// TIA Portal V16 export
// export: Created 2021-11-12T13:32:33.9324246Z, ExportSetting WithDefaults, DisplayName Totally Integrated Automation Portal, DisplayVersion V16 Update 3, DisplayName TIA Portal Version Control Interface, DisplayVersion V16 Update 2, DisplayName TIA Portal Openness, DisplayVersion V16 Update 3, DisplayName SINAMICS Startdrive Advanced, DisplayVersion V16 Update 5, DisplayName SINAMICS Startdrive G130, G150, S120, S150, SINAMICS MV, S210, DisplayVersion V16 Update 5, DisplayName SINAMICS Startdrive G110M, G120, G120C, G120D, G120P, G115D, DisplayVersion V16 Update 5, DisplayName STEP 7 Professional, DisplayVersion V16 Update 3, DisplayName STEP 7 Safety, DisplayVersion V16, DisplayName WinCC UA Professional, DisplayVersion V16 Update 3
FUNCTION_BLOCK "Station220"   // FB16, LAD
{ S7_Optimized_Access := 'TRUE' }
VERSION : 0.1
// Dopravník na ostřižky
// stored: AutoNumber true, IsIECCheckEnabled false, IsRetainMemResEnabled false, MemoryReserve 100, SetENOAutomatically false, UDAEnableTagReadback false
   VAR
      SF_CL01_Alarm { S7_SetPoint := 'True'} : "STD_DI_Mon";
      SF_CL01_Warning { S7_SetPoint := 'True'} : "STD_DI_Mon";
      SF_GL01MA01 { S7_SetPoint := 'True'} : "STD_Drive1";
      SF_UC12TA01 { S7_SetPoint := 'True'} : "STD_Siemens_G120_CU240E_2_PN";
      SF_TON_1 { S7_SetPoint := 'True'} : TON_TIME;
      SF_TOF_1 { S7_SetPoint := 'True'} : TOF_TIME;
      SF_CL01 { S7_SetPoint := 'True'} : "STD_PartCounter";
      SS_Edge { S7_SetPoint := 'True'} : Array[0..15] of Bool;
      SB1BoxExchangeReq { S7_SetPoint := 'True'} : Bool;
   END_VAR
   VAR_TEMP
      TS_GL01MA01 : "UDT_DriveControl";
      TS_UC12TA01 : Struct
         ReqDir1 : Bool;   // Move in direction 1
         ReqDir2 : Bool;   // Move in direction 2
         AckErr : Bool;   // Acknowledge error
         SpeedSP : Real;   // Speed setpoint
      END_STRUCT;
      TB1PwrOK : Bool;
      TDINoOfParts : DInt;   // Number of parts to count
      TB1BoxFull : Bool;   // Box is full
      TB1CountPulse : Bool;
   END_VAR
   VAR_TEMP   // added for the SCL form of the ladder/FBD networks
      _w1 : Bool;
      _w2 : Bool;
      _w3 : Bool;
      _w4 : Bool;
   END_VAR
BEGIN

REGION Network 1: Clear temporary variables
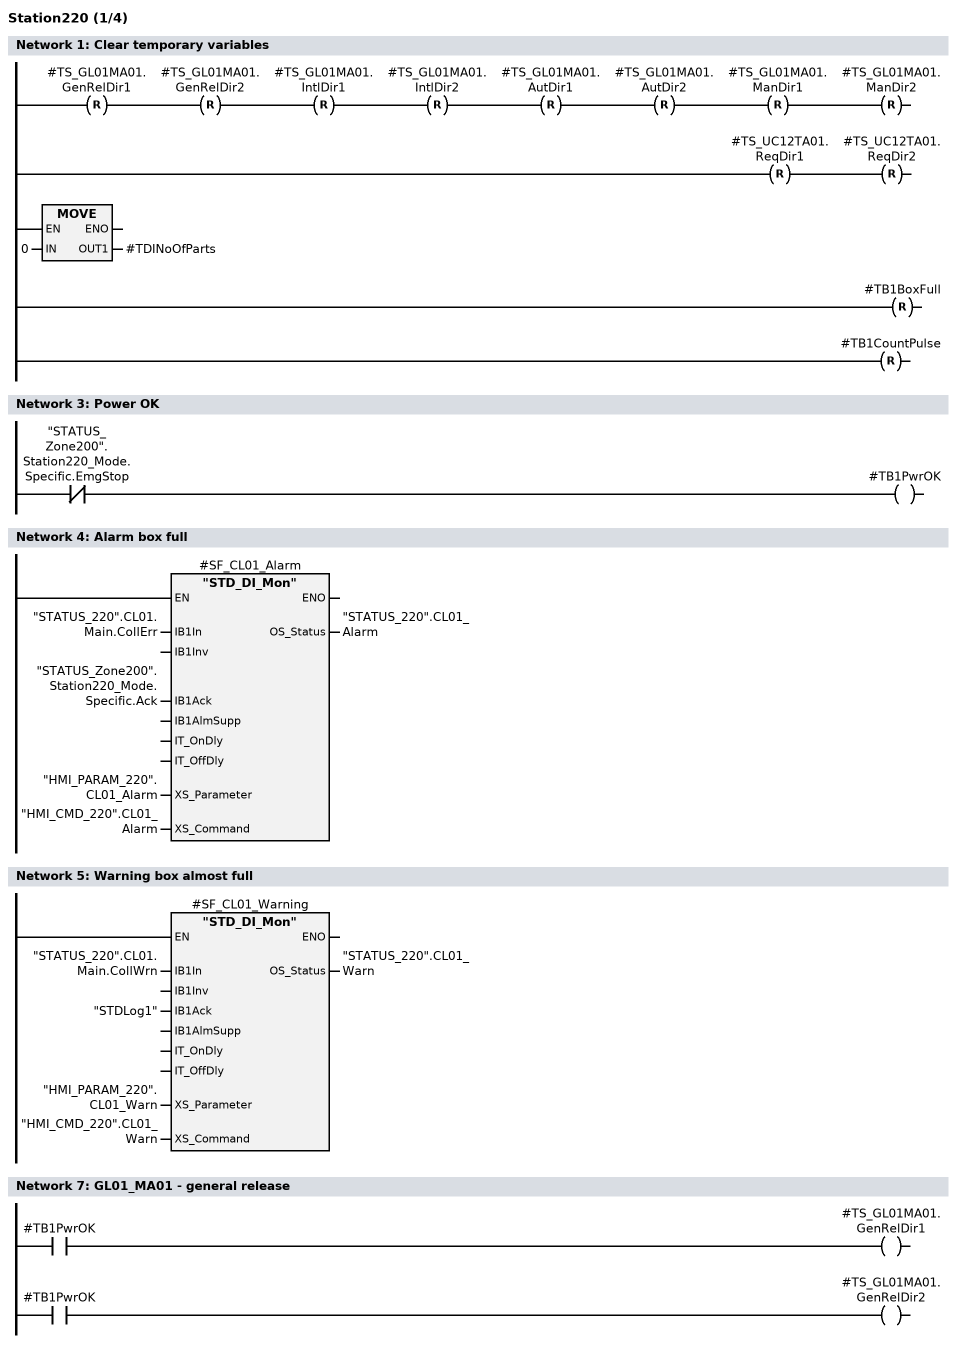
   RUNG wire#powerrail
      R_Coil( #TS_GL01MA01.GenRelDir1 )
      R_Coil( #TS_GL01MA01.GenRelDir2 )
      R_Coil( #TS_GL01MA01.IntlDir1 )
      R_Coil( #TS_GL01MA01.IntlDir2 )
      R_Coil( #TS_GL01MA01.AutDir1 )
      R_Coil( #TS_GL01MA01.AutDir2 )
      R_Coil( #TS_GL01MA01.ManDir1 )
      R_Coil( #TS_GL01MA01.ManDir2 )
   END_RUNG
   RUNG wire#powerrail
      R_Coil( #TS_UC12TA01.ReqDir1 )
      R_Coil( #TS_UC12TA01.ReqDir2 )
   END_RUNG
   RUNG wire#powerrail
      Move(in := 0, out1 => #TDINoOfParts)
   END_RUNG
   RUNG wire#powerrail
      R_Coil( #TB1BoxFull )
   END_RUNG
   RUNG wire#powerrail
      R_Coil( #TB1CountPulse )
   END_RUNG
   // the same network as SCL:
   #TS_GL01MA01.GenRelDir1 := FALSE;
   #TS_GL01MA01.GenRelDir2 := FALSE;
   #TS_GL01MA01.IntlDir1 := FALSE;
   #TS_GL01MA01.IntlDir2 := FALSE;
   #TS_GL01MA01.AutDir1 := FALSE;
   #TS_GL01MA01.AutDir2 := FALSE;
   #TS_GL01MA01.ManDir1 := FALSE;
   #TS_GL01MA01.ManDir2 := FALSE;
   #TS_UC12TA01.ReqDir1 := FALSE;
   #TS_UC12TA01.ReqDir2 := FALSE;
   #TDINoOfParts := 0;
   #TB1BoxFull := FALSE;
   #TB1CountPulse := FALSE;
END_REGION

REGION Network 2: *************** Alarms ***************
END_REGION

REGION Network 3: Power OK
   RUNG wire#powerrail
      I_Contact( "STATUS_Zone200".Station220_Mode.Specific.EmgStop )
      Coil( #TB1PwrOK )
   END_RUNG
   // the same network as SCL:
   #TB1PwrOK := NOT "STATUS_Zone200".Station220_Mode.Specific.EmgStop;
END_REGION

REGION Network 4: Alarm box full
   RUNG wire#powerrail
      #SF_CL01_Alarm(IB1In := "STATUS_220".CL01.Main.CollErr, IB1Inv :=, IB1Ack := "STATUS_Zone200".Station220_Mode.Specific.Ack, IB1AlmSupp :=, IT_OnDly :=, IT_OffDly :=, XS_Parameter := "HMI_PARAM_220".CL01_Alarm, XS_Command := "HMI_CMD_220".CL01_Alarm, OS_Status => "STATUS_220".CL01_Alarm)
   END_RUNG
   // the same network as SCL:
   #SF_CL01_Alarm(IB1In := "STATUS_220".CL01.Main.CollErr,   // "STD_DI_Mon"
                  IB1Ack := "STATUS_Zone200".Station220_Mode.Specific.Ack,
                  XS_Parameter := "HMI_PARAM_220".CL01_Alarm,
                  XS_Command := "HMI_CMD_220".CL01_Alarm,
                  OS_Status => "STATUS_220".CL01_Alarm);
END_REGION

REGION Network 5: Warning box almost full
   RUNG wire#powerrail
      #SF_CL01_Warning(IB1In := "STATUS_220".CL01.Main.CollWrn, IB1Inv :=, IB1Ack := "STDLog1", IB1AlmSupp :=, IT_OnDly :=, IT_OffDly :=, XS_Parameter := "HMI_PARAM_220".CL01_Warn, XS_Command := "HMI_CMD_220".CL01_Warn, OS_Status => "STATUS_220".CL01_Warn)
   END_RUNG
   // the same network as SCL:
   #SF_CL01_Warning(IB1In := "STATUS_220".CL01.Main.CollWrn,   // "STD_DI_Mon"
                    IB1Ack := "STDLog1",
                    XS_Parameter := "HMI_PARAM_220".CL01_Warn,
                    XS_Command := "HMI_CMD_220".CL01_Warn,
                    OS_Status => "STATUS_220".CL01_Warn);
END_REGION

REGION Network 6: *************** GL01_MA01 Conveyor drive ***************
END_REGION

REGION Network 7: GL01_MA01 - general release
   RUNG wire#powerrail
      Contact( #TB1PwrOK )
      Coil( #TS_GL01MA01.GenRelDir1 )
   END_RUNG
   RUNG wire#powerrail
      Contact( #TB1PwrOK )
      Coil( #TS_GL01MA01.GenRelDir2 )
   END_RUNG
   // the same network as SCL:
   #TS_GL01MA01.GenRelDir1 := #TB1PwrOK;
   #TS_GL01MA01.GenRelDir2 := #TB1PwrOK;
END_REGION

REGION Network 8: GL01_MA01 - interlocks
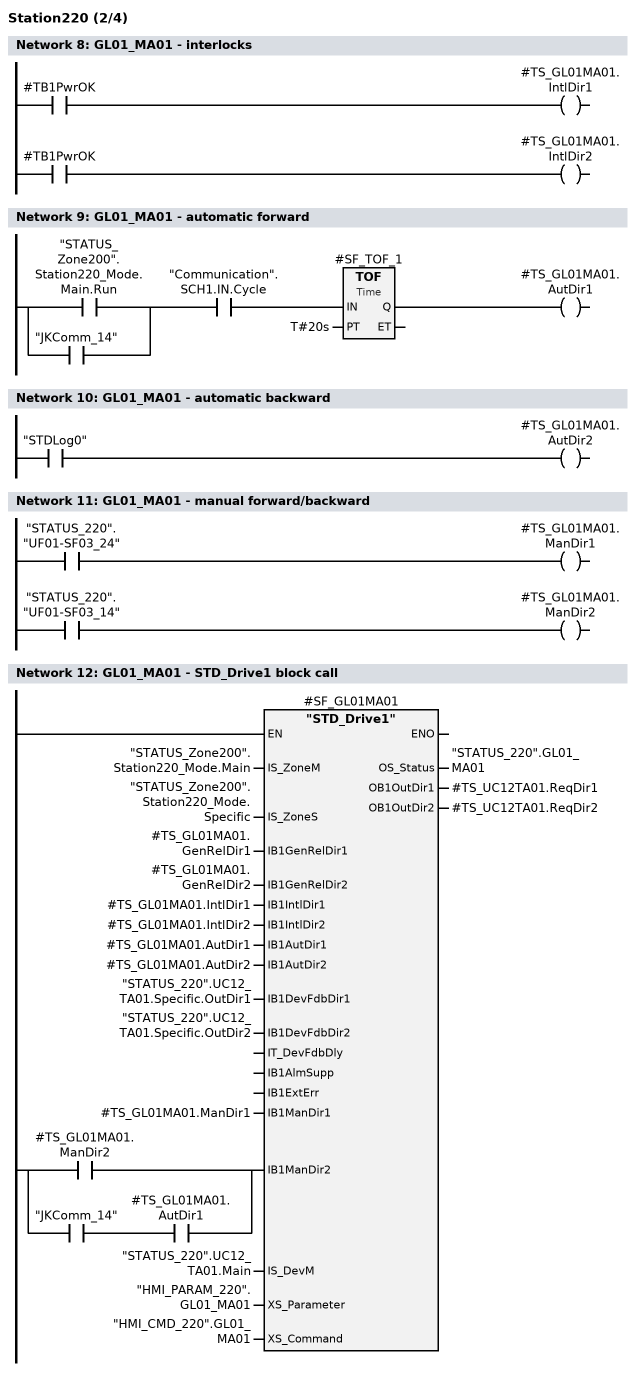
   RUNG wire#powerrail
      Contact( #TB1PwrOK )
      Coil( #TS_GL01MA01.IntlDir1 )
   END_RUNG
   RUNG wire#powerrail
      Contact( #TB1PwrOK )
      Coil( #TS_GL01MA01.IntlDir2 )
   END_RUNG
   // the same network as SCL:
   #TS_GL01MA01.IntlDir1 := #TB1PwrOK;
   #TS_GL01MA01.IntlDir2 := #TB1PwrOK;
END_REGION

REGION Network 9: GL01_MA01 - automatic forward
   RUNG wire#powerrail
      Contact( "STATUS_Zone200".Station220_Mode.Main.Run )
      wire#w1
      Contact( "Communication".SCH1.IN.Cycle )
      { S7_Templates := "time_type := Time" } #SF_TOF_1.TOF(pt := T#20s, et =>)
      Coil( #TS_GL01MA01.AutDir1 )
   END_RUNG
   RUNG wire#powerrail
      Contact( "JKComm_14" )
   END_RUNG wire#w1
   // the same network as SCL:
   #SF_TOF_1(IN := ("STATUS_Zone200".Station220_Mode.Main.Run OR "JKComm_14") AND "Communication".SCH1.IN.Cycle,   // TOF
             PT := T#20s);
   #TS_GL01MA01.AutDir1 := #SF_TOF_1.Q;
END_REGION

REGION Network 10: GL01_MA01 - automatic backward
   RUNG wire#powerrail
      Contact( "STDLog0" )
      Coil( #TS_GL01MA01.AutDir2 )
   END_RUNG
   // the same network as SCL:
   #TS_GL01MA01.AutDir2 := "STDLog0";
END_REGION

REGION Network 11: GL01_MA01 - manual forward/backward
   RUNG wire#powerrail
      Contact( "STATUS_220"."UF01-SF03_24" )
      Coil( #TS_GL01MA01.ManDir1 )
   END_RUNG
   RUNG wire#powerrail
      Contact( "STATUS_220"."UF01-SF03_14" )
      Coil( #TS_GL01MA01.ManDir2 )
   END_RUNG
   // the same network as SCL:
   #TS_GL01MA01.ManDir1 := "STATUS_220"."UF01-SF03_24";
   #TS_GL01MA01.ManDir2 := "STATUS_220"."UF01-SF03_14";
END_REGION

REGION Network 12: GL01_MA01 - STD_Drive1 block call
   RUNG wire#powerrail
      #SF_GL01MA01(IB1ManDir2 := wire#w1, IS_ZoneM := "STATUS_Zone200".Station220_Mode.Main, IS_ZoneS := "STATUS_Zone200".Station220_Mode.Specific, IB1GenRelDir1 := #TS_GL01MA01.GenRelDir1, IB1GenRelDir2 := #TS_GL01MA01.GenRelDir2, IB1IntlDir1 := #TS_GL01MA01.IntlDir1, IB1IntlDir2 := #TS_GL01MA01.IntlDir2, IB1AutDir1 := #TS_GL01MA01.AutDir1, IB1AutDir2 := #TS_GL01MA01.AutDir2, IB1DevFdbDir1 := "STATUS_220".UC12_TA01.Specific.OutDir1, IB1DevFdbDir2 := "STATUS_220".UC12_TA01.Specific.OutDir2, IT_DevFdbDly :=, IB1AlmSupp :=, IB1ExtErr :=, IB1ManDir1 := #TS_GL01MA01.ManDir1, IS_DevM := "STATUS_220".UC12_TA01.Main, XS_Parameter := "HMI_PARAM_220".GL01_MA01, XS_Command := "HMI_CMD_220".GL01_MA01, OS_Status => "STATUS_220".GL01_MA01, OB1OutDir1 => #TS_UC12TA01.ReqDir1, OB1OutDir2 => #TS_UC12TA01.ReqDir2)
   END_RUNG
   RUNG wire#powerrail
      Contact( #TS_GL01MA01.ManDir2 )
   END_RUNG wire#w1
   RUNG wire#powerrail
      Contact( "JKComm_14" )
      Contact( #TS_GL01MA01.AutDir1 )
   END_RUNG wire#w1
   // the same network as SCL:
   #SF_GL01MA01(IS_ZoneM := "STATUS_Zone200".Station220_Mode.Main,   // "STD_Drive1"
                IS_ZoneS := "STATUS_Zone200".Station220_Mode.Specific,
                IB1GenRelDir1 := #TS_GL01MA01.GenRelDir1,
                IB1GenRelDir2 := #TS_GL01MA01.GenRelDir2,
                IB1IntlDir1 := #TS_GL01MA01.IntlDir1,
                IB1IntlDir2 := #TS_GL01MA01.IntlDir2,
                IB1AutDir1 := #TS_GL01MA01.AutDir1,
                IB1AutDir2 := #TS_GL01MA01.AutDir2,
                IB1DevFdbDir1 := "STATUS_220".UC12_TA01.Specific.OutDir1,
                IB1DevFdbDir2 := "STATUS_220".UC12_TA01.Specific.OutDir2,
                IB1ManDir1 := #TS_GL01MA01.ManDir1,
                IB1ManDir2 := #TS_GL01MA01.ManDir2 OR ("JKComm_14" AND #TS_GL01MA01.AutDir1),
                IS_DevM := "STATUS_220".UC12_TA01.Main,
                XS_Parameter := "HMI_PARAM_220".GL01_MA01,
                XS_Command := "HMI_CMD_220".GL01_MA01,
                OS_Status => "STATUS_220".GL01_MA01,
                OB1OutDir1 => #TS_UC12TA01.ReqDir1,
                OB1OutDir2 => #TS_UC12TA01.ReqDir2);
END_REGION

REGION Network 13: UC12_TA01 - Acknowledge error
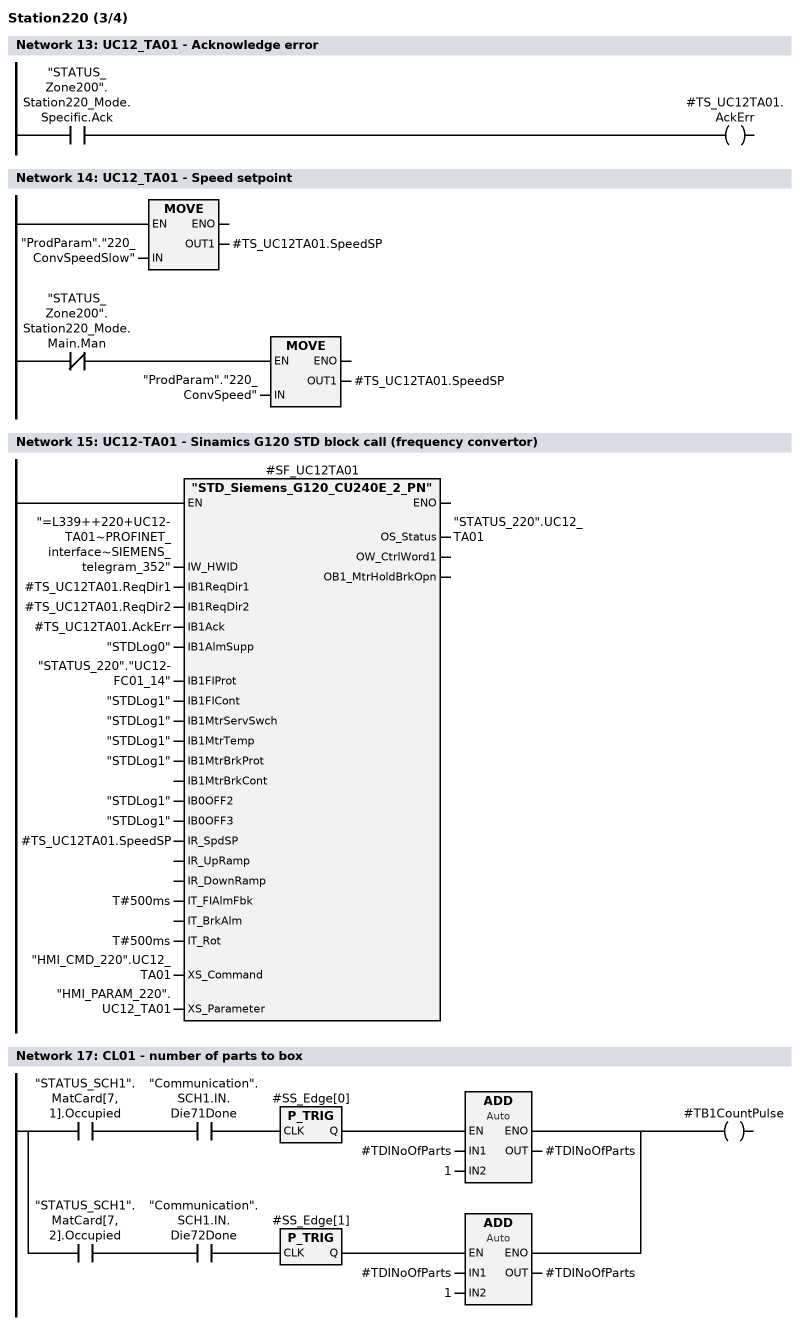
   RUNG wire#powerrail
      Contact( "STATUS_Zone200".Station220_Mode.Specific.Ack )
      Coil( #TS_UC12TA01.AckErr )
   END_RUNG
   // the same network as SCL:
   #TS_UC12TA01.AckErr := "STATUS_Zone200".Station220_Mode.Specific.Ack;
END_REGION

REGION Network 14: UC12_TA01 - Speed setpoint
   RUNG wire#powerrail
      Move(in := "ProdParam"."220_ConvSpeedSlow", out1 => #TS_UC12TA01.SpeedSP)
   END_RUNG
   RUNG wire#powerrail
      I_Contact( "STATUS_Zone200".Station220_Mode.Main.Man )
      Move(in := "ProdParam"."220_ConvSpeed", out1 => #TS_UC12TA01.SpeedSP)
   END_RUNG
   // the same network as SCL:
   #TS_UC12TA01.SpeedSP := "ProdParam"."220_ConvSpeedSlow";
   IF NOT "STATUS_Zone200".Station220_Mode.Main.Man THEN
       #TS_UC12TA01.SpeedSP := "ProdParam"."220_ConvSpeed";
   END_IF;
END_REGION

REGION Network 15: UC12-TA01 - Sinamics G120 STD block call (frequency convertor)
   RUNG wire#powerrail
      #SF_UC12TA01(IW_HWID := "=L339++220+UC12-TA01~PROFINET_interface~SIEMENS_telegram_352", IB1ReqDir1 := #TS_UC12TA01.ReqDir1, IB1ReqDir2 := #TS_UC12TA01.ReqDir2, IB1Ack := #TS_UC12TA01.AckErr, IB1AlmSupp := "STDLog0", IB1FIProt := "STATUS_220"."UC12-FC01_14", IB1FICont := "STDLog1", IB1MtrServSwch := "STDLog1", IB1MtrTemp := "STDLog1", IB1MtrBrkProt := "STDLog1", IB1MtrBrkCont :=, IB0OFF2 := "STDLog1", IB0OFF3 := "STDLog1", IR_SpdSP := #TS_UC12TA01.SpeedSP, IR_UpRamp :=, IR_DownRamp :=, IT_FIAlmFbk := T#500ms, IT_BrkAlm :=, IT_Rot := T#500ms, XS_Command := "HMI_CMD_220".UC12_TA01, XS_Parameter := "HMI_PARAM_220".UC12_TA01, OS_Status => "STATUS_220".UC12_TA01, OW_CtrlWord1 =>, OB1_MtrHoldBrkOpn =>)
   END_RUNG
   // the same network as SCL:
   #SF_UC12TA01(IW_HWID := "=L339++220+UC12-TA01~PROFINET_interface~SIEMENS_telegram_352",   // "STD_Siemens_G120_CU240E_2_PN"
                IB1ReqDir1 := #TS_UC12TA01.ReqDir1,
                IB1ReqDir2 := #TS_UC12TA01.ReqDir2,
                IB1Ack := #TS_UC12TA01.AckErr,
                IB1AlmSupp := "STDLog0",
                IB1FIProt := "STATUS_220"."UC12-FC01_14",
                IB1FICont := "STDLog1",
                IB1MtrServSwch := "STDLog1",
                IB1MtrTemp := "STDLog1",
                IB1MtrBrkProt := "STDLog1",
                IB0OFF2 := "STDLog1",
                IB0OFF3 := "STDLog1",
                IR_SpdSP := #TS_UC12TA01.SpeedSP,
                IT_FIAlmFbk := T#500ms,
                IT_Rot := T#500ms,
                XS_Command := "HMI_CMD_220".UC12_TA01,
                XS_Parameter := "HMI_PARAM_220".UC12_TA01,
                OS_Status => "STATUS_220".UC12_TA01);
END_REGION

REGION Network 16: *************** Box CL01 ***************
END_REGION

REGION Network 17: CL01 - number of parts to box
   RUNG wire#powerrail
      Contact( "STATUS_SCH1".MatCard[7, 1].Occupied )
      Contact( "Communication".SCH1.IN.Die71Done )
      P_Trig( #SS_Edge[0] )
      Add(in1 := #TDINoOfParts, in2 := 1, out => #TDINoOfParts)
      wire#w1
      Coil( #TB1CountPulse )
   END_RUNG
   RUNG wire#powerrail
      Contact( "STATUS_SCH1".MatCard[7, 2].Occupied )
      Contact( "Communication".SCH1.IN.Die72Done )
      P_Trig( #SS_Edge[1] )
      Add(in1 := #TDINoOfParts, in2 := 1, out => #TDINoOfParts)
   END_RUNG wire#w1
   // the same network as SCL:
   #_w1 := "STATUS_SCH1".MatCard[7, 1].Occupied AND "Communication".SCH1.IN.Die71Done;
   #_w2 := #_w1 AND NOT #SS_Edge[0];   // rising edge
   #SS_Edge[0] := #_w1;
   IF #_w2 THEN #TDINoOfParts := #TDINoOfParts + 1; END_IF;
   #_w3 := "STATUS_SCH1".MatCard[7, 2].Occupied AND "Communication".SCH1.IN.Die72Done;
   #_w4 := #_w3 AND NOT #SS_Edge[1];   // rising edge
   #SS_Edge[1] := #_w3;
   IF #_w4 THEN #TDINoOfParts := #TDINoOfParts + 1; END_IF;
   #TB1CountPulse := #_w2 OR #_w4;
END_REGION

REGION Network 18: CL01 - Part counter
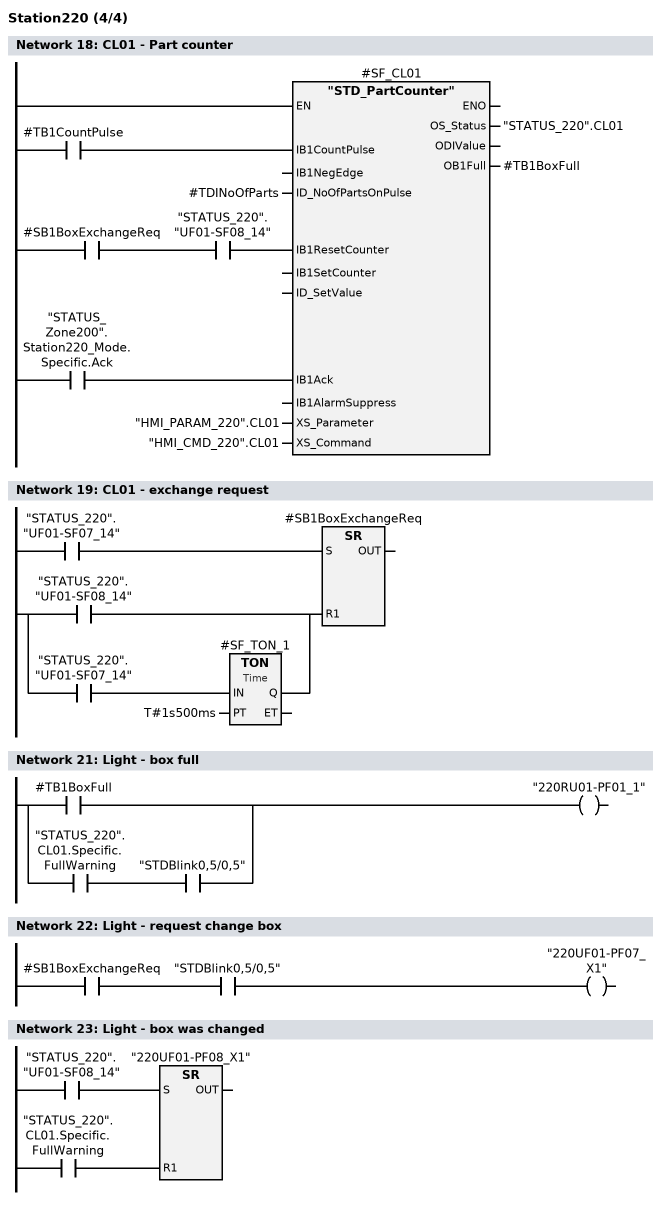
   RUNG wire#powerrail
      #SF_CL01(IB1CountPulse := wire#w1, IB1ResetCounter := wire#w2, IB1Ack := wire#w3, IB1NegEdge :=, ID_NoOfPartsOnPulse := #TDINoOfParts, IB1SetCounter :=, ID_SetValue :=, IB1AlarmSuppress :=, XS_Parameter := "HMI_PARAM_220".CL01, XS_Command := "HMI_CMD_220".CL01, OS_Status => "STATUS_220".CL01, ODIValue =>, OB1Full => #TB1BoxFull)
   END_RUNG
   RUNG wire#powerrail
      Contact( #TB1CountPulse )
   END_RUNG wire#w1
   RUNG wire#powerrail
      Contact( #SB1BoxExchangeReq )
      Contact( "STATUS_220"."UF01-SF08_14" )
   END_RUNG wire#w2
   RUNG wire#powerrail
      Contact( "STATUS_Zone200".Station220_Mode.Specific.Ack )
   END_RUNG wire#w3
   // the same network as SCL:
   #SF_CL01(IB1CountPulse := #TB1CountPulse,   // "STD_PartCounter"
            ID_NoOfPartsOnPulse := #TDINoOfParts,
            IB1ResetCounter := #SB1BoxExchangeReq AND "STATUS_220"."UF01-SF08_14",
            IB1Ack := "STATUS_Zone200".Station220_Mode.Specific.Ack,
            XS_Parameter := "HMI_PARAM_220".CL01,
            XS_Command := "HMI_CMD_220".CL01,
            OS_Status => "STATUS_220".CL01,
            OB1Full => #TB1BoxFull);
END_REGION

REGION Network 19: CL01 - exchange request
   RUNG wire#powerrail
      Contact( "STATUS_220"."UF01-SF07_14" )
      S_SR(operand := #SB1BoxExchangeReq, r1 := wire#w1)
   END_RUNG
   RUNG wire#powerrail
      Contact( "STATUS_220"."UF01-SF08_14" )
   END_RUNG wire#w1
   RUNG wire#powerrail
      Contact( "STATUS_220"."UF01-SF07_14" )
      { S7_Templates := "time_type := Time" } #SF_TON_1.TON(pt := T#1s500ms, et =>)
   END_RUNG wire#w1
   // the same network as SCL:
   #SF_TON_1(IN := "STATUS_220"."UF01-SF07_14", PT := T#1s500ms);   // TON
   IF "STATUS_220"."UF01-SF07_14" THEN
       #SB1BoxExchangeReq := TRUE;   // SR flip-flop
   END_IF;
   IF "STATUS_220"."UF01-SF08_14" OR #SF_TON_1.Q THEN #SB1BoxExchangeReq := FALSE; END_IF;
END_REGION

REGION Network 20: *************** Signalization ***************
END_REGION

REGION Network 21: Light - box full
   RUNG wire#powerrail
      Contact( #TB1BoxFull )
      wire#w1
      Coil( "220RU01-PF01_1" )
   END_RUNG
   RUNG wire#powerrail
      Contact( "STATUS_220".CL01.Specific.FullWarning )
      Contact( "STDBlink0,5/0,5" )
   END_RUNG wire#w1
   // the same network as SCL:
   "220RU01-PF01_1" := #TB1BoxFull OR ("STATUS_220".CL01.Specific.FullWarning AND "STDBlink0,5/0,5");
END_REGION

REGION Network 22: Light - request change box
   RUNG wire#powerrail
      Contact( #SB1BoxExchangeReq )
      Contact( "STDBlink0,5/0,5" )
      Coil( "220UF01-PF07_X1" )
   END_RUNG
   // the same network as SCL:
   "220UF01-PF07_X1" := #SB1BoxExchangeReq AND "STDBlink0,5/0,5";
END_REGION

REGION Network 23: Light - box was changed
   RUNG wire#powerrail
      Contact( "STATUS_220"."UF01-SF08_14" )
      S_SR(operand := "220UF01-PF08_X1", r1 := wire#w1)
   END_RUNG
   RUNG wire#powerrail
      Contact( "STATUS_220".CL01.Specific.FullWarning )
   END_RUNG wire#w1
   // the same network as SCL:
   IF "STATUS_220"."UF01-SF08_14" THEN
       "220UF01-PF08_X1" := TRUE;   // SR flip-flop
   END_IF;
   IF "STATUS_220".CL01.Specific.FullWarning THEN "220UF01-PF08_X1" := FALSE; END_IF;
END_REGION
END_FUNCTION_BLOCK
